// TwinCAT 3 PLC project PLC_Local
// ProgramVersion: 3.1.4026.25
// libraries:
//   Tc2_Standard, * (Beckhoff Automation GmbH)
//   Tc2_System, * (Beckhoff Automation GmbH)
// project tree:
//   DUTs/ ST_SensorData.TcDUT
//   / PlcTask.TcTTO
//   POUs/ MAIN.TcPOU
// real-time tasks:
//   TASK PlcTask: cycle T#10ms, priority 20, ADS port 350

CONFIGURATION PLC_Local
    RESOURCE PLC ON TwinCAT3
        TASK PlcTask(INTERVAL := T#10ms, PRIORITY := 20);
        PROGRAM MAIN WITH PlcTask : MAIN;
    END_RESOURCE
END_CONFIGURATION

// ---- DUTs/ST_SensorData.TcDUT
TYPE ST_SensorData :
STRUCT
    bActive : BOOL;
    nId     : INT;
    fValue  : REAL;
    sName   : STRING(80);        
    aValues : ARRAY[0..4] OF INT;
END_STRUCT
END_TYPE

// ---- POUs/MAIN.TcPOU
PROGRAM MAIN
VAR
	stSensor : ST_SensorData;
    aBuffer  : ARRAY[0..9] OF DINT;
END_VAR

END_PROGRAM
